(* PLC project Unnamed, Unknown Unnamed 1 *)
(* stored: creationDateTime 2023-03-10T10:37:17, modificationDateTime 2023-03-15T15:56:42 *)

(* 978-3-658-16137-8, Aufgabe 2.39 *)
FUNCTION_BLOCK KV_Diagram_optimized_Chart
  VAR_INPUT
    INa : BOOL;
    INb : BOOL;
    INc : BOOL;
    INd : BOOL;
  END_VAR
  VAR_OUTPUT
    OUT1 : BOOL;
    OUT2 : BOOL;
  END_VAR

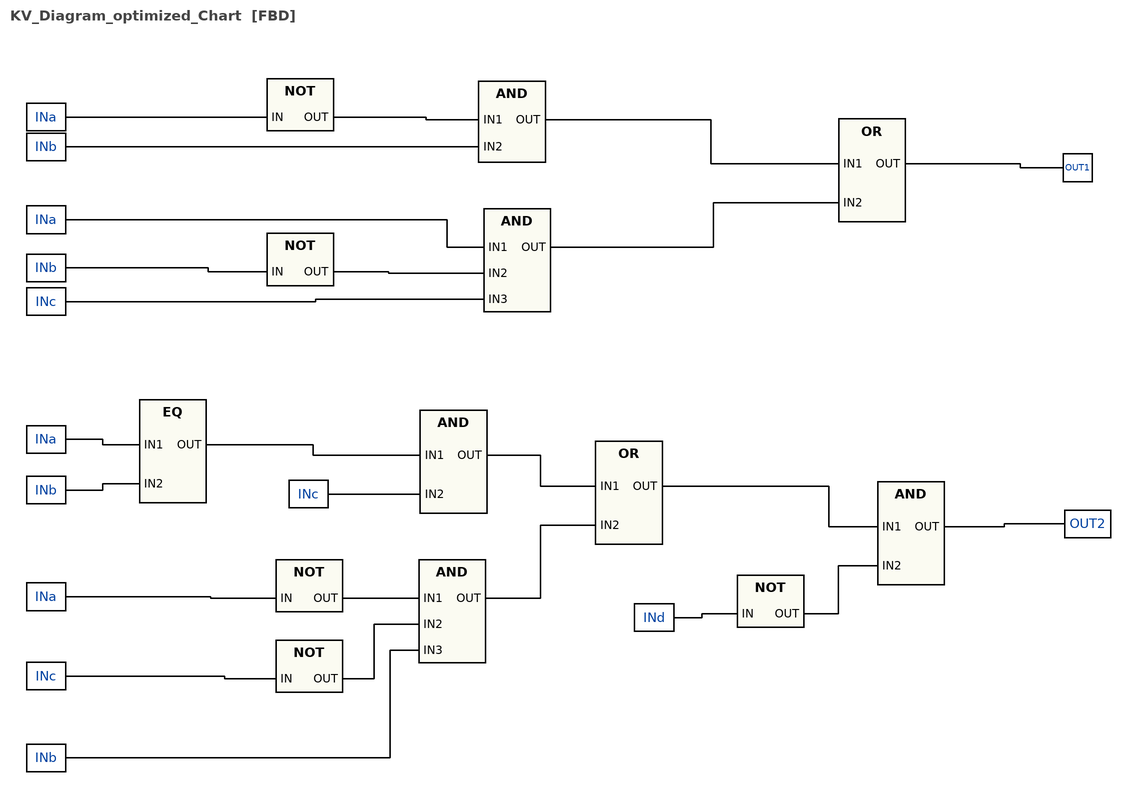
(* FBD diagram, written out as Structured Text *)
OUT1 := NOT INa AND INb OR INa AND NOT INb AND INc;
OUT2 := (INa = INb AND INc OR NOT INa AND NOT INc AND INb) AND NOT INd;
END_FUNCTION_BLOCK

CONFIGURATION config
  RESOURCE resource1 ON PLC
  END_RESOURCE
END_CONFIGURATION
